// Mitsubishi GX Works2 project: sequential counter   PLC: FX1N/FX1NC

PROGRAM MAIN
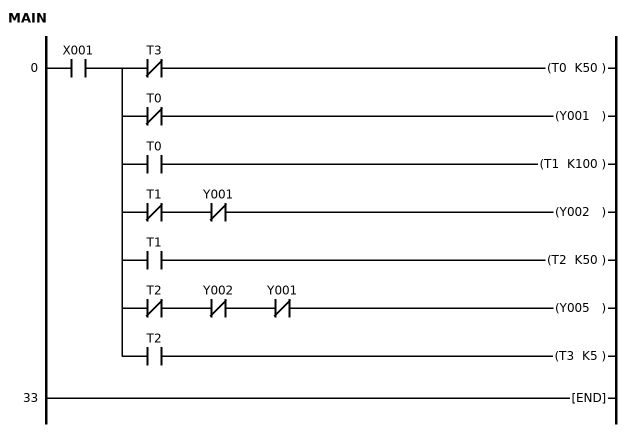
0     LD      X001
      MPS
      ANI     T3
      OUT     T0 K50
      MRD
      ANI     T0
      OUT     Y001
      MRD
      AND     T0
      OUT     T1 K100
      MRD
      ANI     T1
      ANI     Y001
      OUT     Y002
      MRD
      AND     T1
      OUT     T2 K50
      MRD
      ANI     T2
      ANI     Y002
      ANI     Y001
      OUT     Y005
      MPP
      AND     T2
      OUT     T3 K5
33    END
END_PROGRAM
